PROGRAM prgCom
VAR
	fbCom			: FB_MqttCommunicator_V3;
END_VAR

fbCom(
	bConnect:= TRUE, 
	strAuthKey := 'TSG88376368072',
	sUserName:= 'ca71f0f9-cae6-4cad-80bf-5527c253e37c', 
	sUserPassword:= '303ecee9-d411-462e-aea0-ef113d997a29', 
	eSavePositionCertificate:= eSavePositionOnPLC.ePostionC,
	bConnected=> , 
	bError=> , 
	hrErrorCode=> , 
	eConnectionState=> , 
	eErrorMessage_Out=> );

END_PROGRAM

(* stored: Version 1.1.0.1, ProductVersion 3.1.4024.12
   POU prgCom: Id {ab2e2113-e5ef-4576-b3e1-d9e4709b48fc}, SpecialFunc None *)
